# EPICS substitutions: modules/event/evrIoc/Db/evrPatternXL09.substitutions
#
# Pattern records
file evrPatternAll.db
{
#	    Device        ,SLC Pattern
#	                   Check LNK
  pattern { DEVICE        ,LINK4,LINK5,      LINK6         ,  TREF  , TS1ST, TS2ND }
	  { IOC:XL09:EV01 , ""  , ""  ,"BPMS:XX09:1:EFX PP", 1.03E06,   1  ,   4   }
}
# Event records
file evrEventAll.db
{
  pattern { DEVICE        }
	  { IOC:XL09:EV01 }
}
